TYPE EL1008 :
STRUCT
	// 8ch. Digital Input Slot
	e1008	AT %I*	: BYTE;
END_STRUCT
END_TYPE

(* stored: Version 1.1.0.1, ProductVersion 3.1.4024.12
   DUT EL1008: Id {1e4cbd67-7cf4-43f4-a978-10801503e0f1} *)
